ABB RobotStudio station: RoboticsLab1Part2_fazer_de_novo.rspag

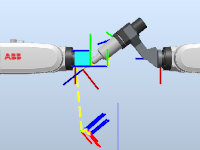
--- station ---
Station RoboticsLab1Part2_2 (saved by RobotStudio 7.0.8732.594)
Controller MMove_System, task T_ROB2: task frame (RAPID world) sits at (-500, 0, 0) mm in the station
Controller MMove_System, task T_ROB1: task frame (RAPID world) sits at (-500, 0, 0) mm in the station
Controller MMove_System
  mechanical unit ROB_1: obj_robot, 6 joints, base frame (0, 0, 0) mm
  mechanical unit ROB_2: tool_robot, 6 joints, base frame (1000, 0, 0) mm, rotated rx 0 ry 0 rz 180 deg
Layout (positions relative to the parent item):
  - tool_robot [mechanism, from Robots\IRB120_3_58_G_01.rslib] at (500, 0, 0) mm, rotated rx 0 ry 0 rz 180 deg; joint values [0, 0, 0, 0, 0, 0] (rad or m)
  - obj_robot [mechanism, from Robots\IRB120_3_58_G_01.rslib] at (-500, 0, 0) mm; joint values [0, 0, 0, 0, 0, 0] (rad or m)
  - MyTool [mechanism, from Training Objects\myTool.rslib] at (126, 0, 630) mm, rotated rx 0 ry 90 rz -180 deg
  - Part_1 [part] at (-126, 0, 630) mm, rotated rx 0 ry 90 rz 0 deg
Attachment: MyTool is attached to tool_robot / Link6
Attachment: Part_1 is attached to obj_robot / Link6
Targets, tools, work objects and paths stored in the station and not in the controller backup, written as RAPID:
! task T_ROB1
MODULE Module1
  VAR SyncIdent Ident_1;
  VAR SyncIdent Ident_2;
ENDMODULE

! task T_ROB2
MODULE Module1
  VAR SyncIdent Ident_1;
  VAR SyncIdent Ident_2;
ENDMODULE


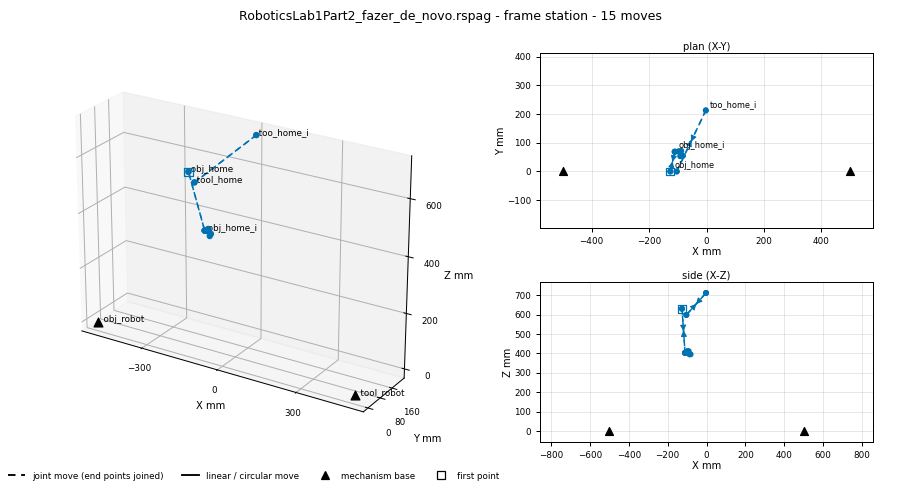
[picture p0: tool path of RoboticsLab1Part2_fazer_de_novo.rspag in frame station, 15 of 29 moves have a stored position in this frame; points joined in program order, loops and branches not executed]
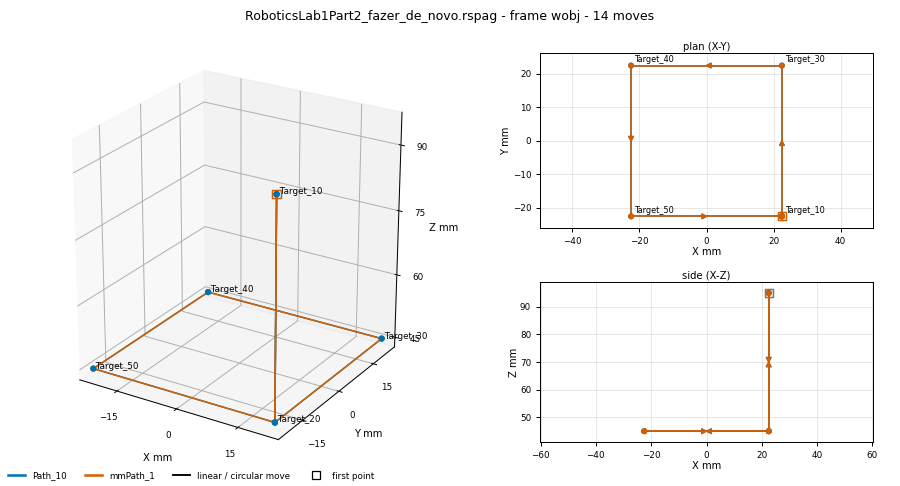
[picture p1: tool path of RoboticsLab1Part2_fazer_de_novo.rspag in frame wobj, 14 of 29 moves have a stored position in this frame; points joined in program order, loops and branches not executed]
--- Backups/MMove_System/RAPID/TASK1/PROGMOD/Module1.mod ---
MODULE Module1
	CONST robtarget obj_home:=[[374,0,630],[0.707106781,0,0.707106781,0],[0,0,0,0],[9E+09,9E+09,9E+09,9E+09,9E+09,9E+09]];
	CONST robtarget obj_home_i:=[[389.564737375,68.799760672,403.063900518],[0.90291697,-0.038025983,0.421324336,0.076031401],[0,0,-1,1],[9E+09,9E+09,9E+09,9E+09,9E+09,9E+09]];
	VAR syncident Ident_1;
	PERS tasks Task_1{2}:=[["T_ROB1"],["T_ROB2"]];
	CONST robtarget pTarget_1:=[[389.240899801,68.63369134,403.647388922],[0.902858991,-0.036833636,0.42101012,0.078989909],[0,0,-1,1],[9E+09,9E+09,9E+09,9E+09,9E+09,9E+09]];
	CONST robtarget pTarget_2:=[[402.452056149,69.796011207,411.713752626],[0.906095131,-0.039925811,0.411987787,0.087542026],[0,-1,0,1],[9E+09,9E+09,9E+09,9E+09,9E+09,9E+09]];
	CONST robtarget pTarget_3:=[[408.40480935,52.996034048,411.605758273],[0.907570219,-0.026518107,0.413424702,0.068506226],[0,-1,0,1],[9E+09,9E+09,9E+09,9E+09,9E+09,9E+09]];
	CONST robtarget pTarget_4:=[[418.184093692,54.644218527,395.460155861],[0.895679586,-0.03056209,0.437397533,0.074212098],[0,-1,0,1],[9E+09,9E+09,9E+09,9E+09,9E+09,9E+09]];
	CONST robtarget pTarget_5:=[[412.099262088,71.70801106,395.484452683],[0.894235579,-0.044721317,0.435774129,0.091889295],[0,-1,0,1],[9E+09,9E+09,9E+09,9E+09,9E+09,9E+09]];
	CONST robtarget pTarget_6:=[[402.75787491,69.959962719,411.178433162],[0.906126228,-0.041101729,0.412435794,0.084514034],[0,-1,0,1],[9E+09,9E+09,9E+09,9E+09,9E+09,9E+09]];
	CONST robtarget pTarget_7:=[[389.564737375,68.799760672,403.063900518],[0.90291697,-0.038025983,0.421324336,0.076031401],[0,0,-1,1],[9E+09,9E+09,9E+09,9E+09,9E+09,9E+09]];
	VAR syncident Ident_2;
    !***********************************************************
    !
    ! Module:  Module1
    !
    ! Description:
    !   <Insert description here>
    !
    ! Author: bruno
    !
    ! Version: 1.0
    !
    !***********************************************************


    !***********************************************************
    !
    ! Procedure main
    !
    !   This is the entry point of your program
    !
    !***********************************************************
    PROC main()
        !Add your code here
    ENDPROC
	PROC mmPath_1()
	    MoveJ obj_home,v1000,z100,tool0\WObj:=wobj0;
	    MoveJ obj_home_i,v1000,z100,tool0\WObj:=wobj0;
	    SyncMoveOn Ident_1,Task_1;
	    MoveL pTarget_1\ID:=10,v1000,z100,tool0\WObj:=wobj0;
	    MoveL pTarget_2\ID:=20,v1000,z100,tool0\WObj:=wobj0;
	    MoveL pTarget_3\ID:=30,v1000,z100,tool0\WObj:=wobj0;
	    MoveL pTarget_4\ID:=40,v1000,z100,tool0\WObj:=wobj0;
	    MoveL pTarget_5\ID:=50,v1000,z100,tool0\WObj:=wobj0;
	    MoveL pTarget_6\ID:=60,v1000,z100,tool0\WObj:=wobj0;
	    MoveL pTarget_7\ID:=70,v1000,fine,tool0\WObj:=wobj0;
	    SyncMoveOff Ident_2;
	    MoveJ obj_home_i,v1000,z100,tool0\WObj:=wobj0;
	    MoveJ obj_home,v1000,z100,tool0\WObj:=wobj0;
	ENDPROC
ENDMODULE

--- Backups/MMove_System/RAPID/TASK2/PROGMOD/CalibData.mod ---
MODULE CalibData
	PERS tooldata MyTool:=[TRUE,[[31.792631019,0,229.638935148],[0.945518576,0,0.325568154,0]],[1,[0,0,1],[1,0,0,0],0,0,0]];
	TASK PERS wobjdata wobj:=[FALSE,FALSE,"ROB_1",[[414.575,-22.5,590.986],[0.353553559,-0.612372339,0.612372339,-0.353553559]],[[0,0,0],[1,0,0,0]]];
ENDMODULE

--- Backups/MMove_System/RAPID/TASK2/PROGMOD/Module1.mod ---
MODULE Module1
	CONST robtarget Target_10:=[[22.5,-22.5,95],[0,-0.707106781,0.707106781,0],[0,0,0,0],[9E+09,9E+09,9E+09,9E+09,9E+09,9E+09]];
	CONST robtarget Target_20:=[[22.5,-22.5,45],[0,-0.707106781,0.707106781,0],[0,0,0,0],[9E+09,9E+09,9E+09,9E+09,9E+09,9E+09]];
	CONST robtarget Target_30:=[[22.5,22.5,45],[0,-0.707106781,0.707106781,0],[0,0,0,0],[9E+09,9E+09,9E+09,9E+09,9E+09,9E+09]];
	CONST robtarget Target_40:=[[-22.5,22.5,45],[0,-0.707106781,0.707106781,0],[0,0,0,0],[9E+09,9E+09,9E+09,9E+09,9E+09,9E+09]];
	CONST robtarget Target_50:=[[-22.5,-22.5,45],[0,-0.707106781,0.707106781,0],[0,0,0,0],[9E+09,9E+09,9E+09,9E+09,9E+09,9E+09]];
	CONST robtarget Target_60:=[[22.5,-22.5,45],[0,-0.707106781,0.707106781,0],[0,0,0,0],[9E+09,9E+09,9E+09,9E+09,9E+09,9E+09]];
	CONST robtarget Target_70:=[[22.5,-22.5,95],[0,-0.707106781,0.707106781,0],[0,0,0,0],[9E+09,9E+09,9E+09,9E+09,9E+09,9E+09]];
	CONST robtarget tool_home:=[[396.361077393,0,598.207406271],[0,0.898794033,0,-0.438371175],[0,0,0,0],[9E+09,9E+09,9E+09,9E+09,9E+09,9E+09]];
	CONST robtarget tool_home_i:=[[497.628534425,-190.861062912,754.177892685],[0.644826216,-0.258593411,-0.374420531,0.614115515],[0,1,1,0],[9E+09,9E+09,9E+09,9E+09,9E+09,9E+09]];
	VAR syncident Ident_1;
	PERS tasks Task_1{2}:=[["T_ROB1"],["T_ROB2"]];
	CONST robtarget pTarget_1:=[[22.5,-22.5,95],[0,-0.707106781,0.707106781,0],[0,-1,1,0],[9E+09,9E+09,9E+09,9E+09,9E+09,9E+09]];
	CONST robtarget pTarget_2:=[[22.5,-22.5,45],[0,-0.707106781,0.707106781,0],[0,-1,1,0],[9E+09,9E+09,9E+09,9E+09,9E+09,9E+09]];
	CONST robtarget pTarget_3:=[[22.5,22.5,45],[0,-0.707106781,0.707106781,0],[0,-1,1,0],[9E+09,9E+09,9E+09,9E+09,9E+09,9E+09]];
	CONST robtarget pTarget_4:=[[-22.5,22.5,45],[0,-0.707106781,0.707106781,0],[0,-1,1,0],[9E+09,9E+09,9E+09,9E+09,9E+09,9E+09]];
	CONST robtarget pTarget_5:=[[-22.5,-22.5,45],[0,-0.707106781,0.707106781,0],[0,-1,1,0],[9E+09,9E+09,9E+09,9E+09,9E+09,9E+09]];
	CONST robtarget pTarget_6:=[[22.5,-22.5,45],[0,-0.707106781,0.707106781,0],[0,-1,1,0],[9E+09,9E+09,9E+09,9E+09,9E+09,9E+09]];
	CONST robtarget pTarget_7:=[[22.5,-22.5,95],[0,-0.707106781,0.707106781,0],[0,-1,1,0],[9E+09,9E+09,9E+09,9E+09,9E+09,9E+09]];
	VAR syncident Ident_2;
	CONST robtarget too_home_i:=[[497.62855396,212.647343524,711.419940513],[0.062336549,-0.691943298,0.377197568,0.612413766],[0,-2,1,0],[9E+09,9E+09,9E+09,9E+09,9E+09,9E+09]];
    !***********************************************************
    !
    ! Module:  Module1
    !
    ! Description:
    !   <Insert description here>
    !
    ! Author: bruno
    !
    ! Version: 1.0
    !
    !***********************************************************


    !***********************************************************
    !
    ! Procedure main
    !
    !   This is the entry point of your program
    !
    !***********************************************************
    PROC main()
        !Add your code here
    ENDPROC
	PROC Path_10()
	    MoveL Target_10,v1000,z100,MyTool\WObj:=wobj;
	    MoveL Target_20,v1000,z100,MyTool\WObj:=wobj;
	    MoveL Target_30,v1000,z100,MyTool\WObj:=wobj;
	    MoveL Target_40,v1000,z100,MyTool\WObj:=wobj;
	    MoveL Target_50,v1000,z100,MyTool\WObj:=wobj;
	    MoveL Target_60,v1000,z100,MyTool\WObj:=wobj;
	    MoveL Target_70,v1000,z100,MyTool\WObj:=wobj;
	ENDPROC
	PROC mmPath_1()
	    MoveJ tool_home,v1000,z100,MyTool\WObj:=wobj0;
	    MoveJ too_home_i,v1000,z100,MyTool\WObj:=wobj0;
	    SyncMoveOn Ident_1,Task_1;
	    MoveJ pTarget_1\ID:=10,v1000,z100,MyTool\WObj:=wobj;
	    MoveL pTarget_2\ID:=20,v1000,z100,MyTool\WObj:=wobj;
	    MoveL pTarget_3\ID:=30,v1000,z100,MyTool\WObj:=wobj;
	    MoveL pTarget_4\ID:=40,v1000,z100,MyTool\WObj:=wobj;
	    MoveL pTarget_5\ID:=50,v1000,z100,MyTool\WObj:=wobj;
	    MoveL pTarget_6\ID:=60,v1000,z100,MyTool\WObj:=wobj;
	    MoveL pTarget_7\ID:=70,v1000,fine,MyTool\WObj:=wobj;
	    SyncMoveOff Ident_2;
	    MoveJ too_home_i,v1000,z100,MyTool\WObj:=wobj0;
	    MoveJ tool_home,v1000,z100,MyTool\WObj:=wobj0;
	ENDPROC
ENDMODULE
